// TwinCAT 3 PLC project Plc
// ProgramVersion: 3.1.4023.0
// libraries:
//   Tc2_Standard, * (Beckhoff Automation GmbH)
//   Tc2_System, * (Beckhoff Automation GmbH)
//   Tc3_Module, * (Beckhoff Automation GmbH)
// project tree:
//   DUTs/ StructWith5Variables.TcDUT, StructWith68Variables.TcDUT, StructWith50Variables.TcDUT
//   / PlcTask.TcTTO
//   POUs/ MAIN.TcPOU
// real-time tasks:
//   TASK PlcTask: cycle T#10ms, priority 20, ADS port 350

CONFIGURATION Plc
    RESOURCE PLC ON TwinCAT3
        TASK PlcTask(INTERVAL := T#10ms, PRIORITY := 20);
        PROGRAM MAIN WITH PlcTask : MAIN;
    END_RESOURCE
END_CONFIGURATION

// ---- DUTs/StructWith5Variables.TcDUT
TYPE
    StructWith5Variables :
    STRUCT
        Variable1 : INT;
        Variable2 : INT;
        Variable3 : INT;
        Variable4 : INT;
        Variable5 : INT;
    END_STRUCT
END_TYPE

// ---- DUTs/StructWith68Variables.TcDUT
TYPE
    StructWith68Variables :
    STRUCT
        Variable1 : STRING;
        Variable2 : STRING;
        Variable3 : STRING;
        Variable4 : STRING;
        Variable5 : STRING;
        Variable6 : STRING;
        Variable7 : STRING;
        Variable8 : STRING;
        Variable9 : STRING;
        Variable10 : STRING;
        Variable11 : STRING;
        Variable12 : STRING;
        Variable13 : STRING;
        Variable14 : STRING;
        Variable15 : STRING;
        Variable16 : STRING;
        Variable17 : STRING;
        Variable18 : STRING;
        Variable19 : STRING;
        Variable20 : STRING;
        Variable21 : STRING;
        Variable22 : STRING;
        Variable23 : STRING;
        Variable24 : STRING;
        Variable25 : STRING;
        Variable26 : STRING;
        Variable27 : STRING;
        Variable28 : STRING;
        Variable29 : STRING;
        Variable30 : STRING;
        Variable31 : STRING;
        Variable32 : STRING;
        Variable33 : STRING;
        Variable34 : STRING;
        Variable35 : STRING;
        Variable36 : STRING;
        Variable37 : STRING;
        Variable38 : STRING;
        Variable39 : STRING;
        Variable40 : STRING;
        Variable41 : STRING;
        Variable42 : STRING;
        Variable43 : STRING;
        Variable44 : STRING;
        Variable45 : STRING;
        Variable46 : STRING;
        Variable47 : STRING;
        Variable48 : STRING;
        Variable49 : STRING;
        Variable50 : STRING;
        Variable51 : STRING;
        Variable52 : STRING;
        Variable53 : STRING;
        Variable54 : STRING;
        Variable55 : STRING;
        Variable56 : STRING;
        Variable57 : STRING;
        Variable58 : STRING;
        Variable59 : STRING;
        Variable60 : STRING;
        Variable61 : STRING;
        Variable62 : STRING;
        Variable63 : STRING;
        Variable64 : STRING;
        Variable65 : STRING;
        Variable66 : STRING;
        Variable67 : STRING;
        Variable68 : STRING;
    END_STRUCT
END_TYPE

// ---- DUTs/StructWith50Variables.TcDUT
TYPE
    StructWith50Variables :
    STRUCT
        Variable1 : INT;
        Variable2 : INT;
        Variable3 : INT;
        Variable4 : INT;
        Variable5 : INT;
        Variable6 : INT;
        Variable7 : INT;
        Variable8 : INT;
        Variable9 : INT;
        Variable10 : INT;
        Variable11 : INT;
        Variable12 : INT;
        Variable13 : INT;
        Variable14 : INT;
        Variable15 : INT;
        Variable16 : INT;
        Variable17 : INT;
        Variable18 : INT;
        Variable19 : INT;
        Variable20 : INT;
        Variable21 : INT;
        Variable22 : INT;
        Variable23 : INT;
        Variable24 : INT;
        Variable25 : INT;
        Variable26 : INT;
        Variable27 : INT;
        Variable28 : INT;
        Variable29 : INT;
        Variable30 : INT;
        Variable31 : INT;
        Variable32 : INT;
        Variable33 : INT;
        Variable34 : INT;
        Variable35 : INT;
        Variable36 : INT;
        Variable37 : INT;
        Variable38 : INT;
        Variable39 : INT;
        Variable40 : INT;
        Variable41 : INT;
        Variable42 : INT;
        Variable43 : INT;
        Variable44 : INT;
        Variable45 : INT;
        Variable46 : INT;
        Variable47 : INT;
        Variable48 : INT;
        Variable49 : INT;
        Variable50 : INT;
    END_STRUCT
END_TYPE

// ---- POUs/MAIN.TcPOU
PROGRAM MAIN
VAR
	first : StructWith50Variables;
	second : StructWith5Variables;
	third : StructWith68Variables;
	
	
	ShouldBe5 : INT;
	ShouldBe68 :INT;
	ShouldBe50 :INT; 
END_VAR

//external programm will write to variables ShouldBe5, ShouldBe68, ShouldBe50

END_PROGRAM
